{attribute 'linkalways'} 
{attribute 'no_explicit_call' := 'This FB is a CLASS and must be accessed using methods or properties'}
{attribute 'enable_dynamic_creation'}
FUNCTION_BLOCK MockUnitMode EXTENDS DefaultUnitMode<State.Idle>
VAR
END_VAR

METHOD PUBLIC StateComplete
state_machine.StateComplete();
END_METHOD

END_FUNCTION_BLOCK

(* stored: Version 1.1.0.1
   POU MockUnitMode: Id {23f7f16b-0a3d-0438-2fe0-39f9efc55b06}, SpecialFunc None
   Method StateComplete: Id {527ee925-d6c9-01e9-1630-82e9efd9b109} *)
